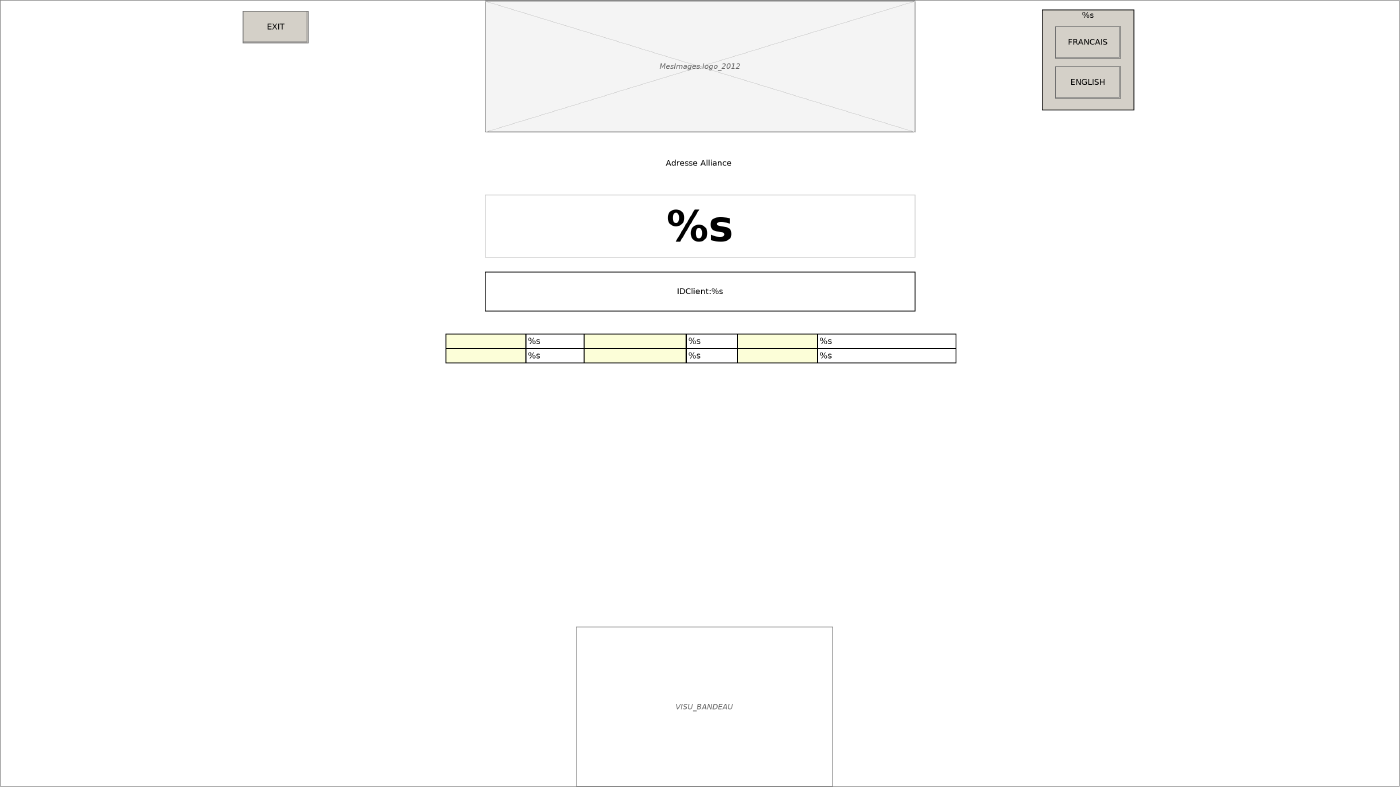
VISUALIZATION SYN_INFOS  // 1920x1080
    Image (665,1 590x180), image: MesImages.logo_2012
    Textfield (665,181 590x86), "Adresse Alliance"
    Textfield (665,267 590x86), "%s", text variable: MACHINE.CONF_Name
    RoundedRectangle (665,373 590x54), "IDClient:%s", text variable: MACHINE.CONF_Customer
    Rectangle (611,458 110x20), text list: 'TextList_Infos', text index: 1
    Rectangle (721,458 80x20), "%s", text variable: Global_Variables.MACHINE.CONF_Affaire
    Rectangle (611,478 110x20), text list: 'TextList_Infos', text index: 2
    Rectangle (721,478 80x20), "%s", text variable: Global_Variables.MACHINE.CONF_Author
    Rectangle (801,478 140x20), text list: 'TextList_Infos', text index: 4
    Rectangle (941,458 70x20), "%s", text variable: Global_Variables.MACHINE.CONF_Version
    Rectangle (801,458 140x20), text list: 'TextList_Infos', text index: 3
    Rectangle (941,478 70x20), "%s", text variable: Global_Variables.MACHINE.CONF_VerDate
    Rectangle (1011,478 110x20), text list: 'TextList_Infos', text index: 6
    Rectangle (1121,458 190x20), "%s", text variable: Global_Variables.MACHINE.CONF_SerialNumber
    Rectangle (1011,458 110x20), text list: 'TextList_Infos', text index: 5
    Rectangle (1121,478 190x20), "%s", text variable: Global_Variables.MACHINE.CONF_Model
    RoundedRectangle (1429,13 126x138), "%s", text list: 'TextList_Infos', text index: 0
    Button (1447,36 90x44), "FRANCAIS"
        OnMouseClick: ChangeLanguage ChangeLanguage=FR
    Button (1447,91 90x44), "ENGLISH"
        OnMouseClick: ChangeLanguage ChangeLanguage=EN
    Frame (790,860 352x220)
        shows VISU_BANDEAU(m_Input_MACHINE := Global_Variables.MACHINE)
    Button (333,15 90x44), "EXIT", text list: ''
        OnMouseClick: change screen: SYN_PROC
        OnMouseDown: ExecuteCommand ExecuteCommand=ExecuteCommand=[Command=ExecuteClientProgram, Value='C:\Machine\PLC\Exit_TC3Hmi.bat']
END_VISUALIZATION

(* stored: Version 1.1.0.1, ProductVersion 3.1.4024.10
   Visu SYN_INFOS: Id {1596b2b6-d013-470b-b975-fdb9e361f170} *)
